{attribute 'qualified_only'}
VAR_GLOBAL
 MHS : ARRAY [1..20] OF DINT;
END_VAR

(* stored: Version 1.1.0.1, ProductVersion 3.1.4024.3
   GVL MHS_Registers: Id {d041caa9-784e-4cfd-97a4-60b9a37cb704} *)
